SUBAPPLICATION logiBUS_IXA_TO_logiBUS_QXA (* logiBUS_IXA auf logiBUS_QXA (generisch) *)
  (* Standard: 61499-2; Description: Copyright (c) 2023 Meisterschulen am Ostbahnhof This program and the accompanying materials are made available under the terms of the Eclipse Public License 2.0 which is available at https://www.eclipse.org/legal/epl-2.0/ SPDX-License-Identifier: EPL-2.0 *)
  (* Version 1.1, 2026-09-18, Franz Höpfinger, Meisterschulen am Ostbahnhof, logiBUS_IXA.INITO auf logiBUS_IXA.REQ zurueckverdrahtet (Selfloop) - loest nach der Initialisierung sofort einen Service-Request aus, statt auf die erste echte Wertaenderung am Bus zu warten (Fix fuer 'Waiting for handle'-Status direkt nach Boot). *)
  (* Version 1.0, 2023-10-23, Franz Höpfinger, Meisterschulen am Ostbahnhof, initial API and implementation and/or initial documentation *)
  PACKAGE MyLib::sys;
  IMPORT logiBUS::io::DI::logiBUS_DI;
  IMPORT logiBUS::io::DI::logiBUS_DI_S;
  IMPORT logiBUS::io::DQ::logiBUS_DO;
  IMPORT logiBUS::io::DQ::logiBUS_DO_S;
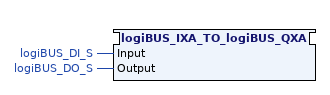
  VAR_INPUT
    Input : logiBUS::io::DI::logiBUS_DI_S := logiBUS_DI::Invalid; (* Identify the Input Input_I1..I8 *)
    Output : logiBUS::io::DQ::logiBUS_DO_S := logiBUS_DO::Invalid; (* Identify the Output Output_Q1..Q8 *)
  END_VAR
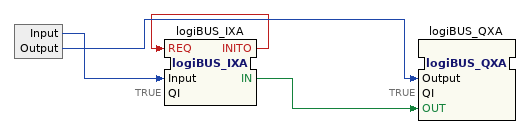
  FBS
    logiBUS_QXA : logiBUS::io::DQ::logiBUS_QXA(QI := TRUE);
    logiBUS_IXA : logiBUS::io::DI::logiBUS_IXA(QI := TRUE);
  END_FBS
  EVENT_CONNECTIONS
    logiBUS_IXA.INITO TO logiBUS_IXA.REQ;
  END_CONNECTIONS
  DATA_CONNECTIONS
    Input TO logiBUS_IXA.Input;
    Output TO logiBUS_QXA.Output;
  END_CONNECTIONS
  ADAPTER_CONNECTIONS
    logiBUS_IXA.IN TO logiBUS_QXA.OUT;
  END_CONNECTIONS
END_SUBAPPLICATION
